TYPE ST_K1100 :
STRUCT
	
	// TERMINAL - K1100	EtherCAT Coupler	 (Term 1)
	sTerminalName                                           :   STRING(200):= 'K1100 | EtherCAT Coupler';
	stTerminalInfo											: 	ST_Terminal_Info;

END_STRUCT
END_TYPE

(* stored: Version 1.1.0.1, ProductVersion 3.1.4024.13
   DUT ST_K1100: Id {8319a722-f9cf-4617-8df3-74065a0d2499} *)
